{attribute 'qualified_only'}
{attribute 'strict'}
{attribute 'to_string'}
TYPE E_MaterialCmdType :
(
	Modify:= 1,
	Clear,
	ClearAll
);
END_TYPE

(* stored: Version 1.1.0.1, ProductVersion 3.1.4026.18
   DUT E_MaterialCmdType: Id {938f2a33-6863-4ddb-baf5-37d09f5fe3f7} *)
